TYPE EtcMasterBase_62654B43 :
STRUCT
END_STRUCT
END_TYPE

(* stored: Version 1.2.0.0, ProductVersion 3.1.4024.11
   DUT EtcMasterBase_62654B43: Id {5860bd87-cdf7-4b1e-85b9-286581bd49e6} *)
